KUKA KRL program: ho_st_60301.src, ho_st_60301.dat

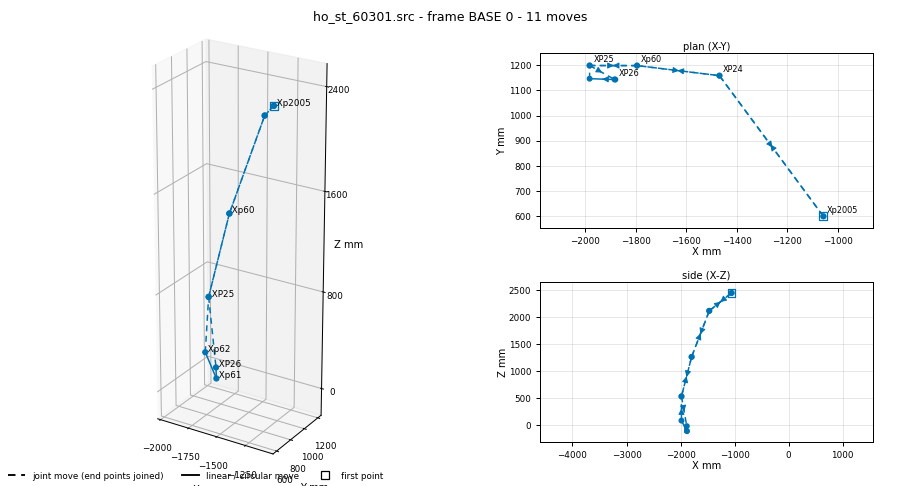
[picture p0: tool path of ho_st_60301.src in frame BASE 0, 11 of 11 moves have a stored position in this frame; points joined in program order, loops and branches not executed]
--- ho_st_60301.src ---
&ACCESS RV2
&REL 251
&COMMENT Busca Peca Frontal Accelo
&PARAM TEMPLATE = C:\KRC\Roboter\Template\vorgabe
&PARAM EDITMASK = *
DEF ho_st_60301( )
;FOLD INI;%{PE}%V3.2.0,%MKUKATPBASIS,%CINIT,%VCOMMON,%P
;FOLD BAS INI;%{E}%V3.2.0,%MKUKATPBASIS,%CINIT,%VINIT,%P
GLOBAL INTERRUPT DECL 3 WHEN $STOPMESS==TRUE DO IR_STOPM ( )
INTERRUPT ON 3
BAS (#INITMOV,0 )
;ENDFOLD (BAS INI)
;FOLD A20 INI;%{E}%V3.2.0,%MKUKATPA20,%CINIT,%VINIT,%P
IF ARC20==TRUE THEN
A20 (ARC_INI)
INTERRUPT DECL 6 WHEN $CYCFLAG[3]==FALSE DO A20(TECH_STOP2)
ENDIF
;ENDFOLD (A20 INI)
;FOLD A10 INI;%{E}%V3.2.0,%MKUKATPARC,%CINIT,%VINIT,%P
IF A10_OPTION==#ACTIVE THEN
INTERRUPT DECL 4 WHEN $CYCFLAG[2]==FALSE DO A10 (#APPL_ERROR)
INTERRUPT DECL 7 WHEN A_ARC_SWI==#ACTIVE DO A10 (#ARC_SEAM)
INTERRUPT DECL 5 WHEN A_FLY_ARC==TRUE DO A10 (#HPU_ARC)
INTERRUPT  ON 5
A10_INI ( )
ENDIF
;ENDFOLD (A10 INI)
;FOLD GRIPPER INI;%{E}%V3.2.0,%MKUKATPGRIPPER,%CINIT,%VINIT,%P
USER_GRP(0,DUMMY,DUMMY,GDEFAULT)
;ENDFOLD (GRIPPER INI)
;FOLD SPOT INI;%{E}%V3.2.0,%MKUKATPSPOT,%CINIT,%VINIT,%P
USERSPOT(#INIT)
;ENDFOLD (SPOT INI)
;FOLD TOUCHSENSE INI;%{E}%V3.2.0,%MKUKATPTS,%CINIT,%VINIT,%P
IF H70_OPTION THEN
INTERRUPT DECL 15 WHEN $MEAS_PULSE[TOUCH_I[TOUCH_ACTIVE].IN_NR] DO H70 (6,CD0 )
INTERRUPT DECL 16 WHEN $ZERO_MOVE DO H70 (7,CD0 )
INTERRUPT DECL 17 WHEN $TECHPAR_C[FG_TOUCH,8]>0.5 DO H70 (8,CD0)
H70 (1,CD0 )
ENDIF
;ENDFOLD (TOUCHSENSE INI)
;FOLD USER INI;%{E}%V3.2.0,%MKUKATPUSER,%CINIT,%VINIT,%P
;Make your modifications here
;ENDFOLD (USER INI)
;ENDFOLD (INI)

; Caracterização dos meios de produção:
; Versão Atual:
; 19/07/2013 12:00 Name: P13.060-R3 CHANGES: Busca Frontal Accelo
; na Geobox

chk_w3_wechs_ok ( )        ;VERIFICAÇÃO DE FERRAMENTA: griper frontal acelo

;FOLD PTP p2005  Vel= 100 % PDAT54 Tool[3]:Gripper Frontal Accelo Base[0];%{PE}%R 4.1.16,%MKUKATPBASIS,%CMOVE,%VPTP,%P 1:PTP, 2:p2005, 3:, 5:100, 7:PDAT54
$BWDSTART = FALSE
PDAT_ACT=PPDAT54
BAS(#PTP_DAT)
FDAT_ACT=Fp2005
BAS(#FRAMES)
BAS(#VEL_PTP,100)
PTP Xp2005
;ENDFOLD

;FOLD OUT 826 'Busca frontal Accelo'  State= TRUE ;%{PE}%R 4.1.16,%MKUKATPBASIS,%COUT,%VOUTX,%P 2:826, 3:'Busca frontal Accelo', 5:TRUE, 6:
$OUT[826]=TRUE
;ENDFOLD
;FOLD OUT 825 'R3 Solic Lib Entrar EST 060 EL_631 '  State= TRUE ;%{PE}%R 4.1.16,%MKUKATPBASIS,%COUT,%VOUTX,%P 2:825, 3:'R3 Solic Lib Entrar EST 060 EL_631 ', 5:TRUE, 6:
$OUT[825]=TRUE
;ENDFOLD
;FOLD WAIT FOR IN 826 'aguarda lib. buscar frontal Accelo'  State= TRUE ;%{PE}%R 4.1.16,%MKUKATPBASIS,%CWAIT_FOR,%VWAIT_FOR,%P 1:0, 2:826, 3:'aguarda lib. buscar frontal Accelo', 5:TRUE, 6:
WAIT FOR $IN[826]==TRUE
;ENDFOLD
;FOLD OUT 826 'Busca frontal Accelo'  State= FALSE ;%{PE}%R 4.1.16,%MKUKATPBASIS,%COUT,%VOUTX,%P 2:826, 3:'Busca frontal Accelo', 5:FALSE, 6:
$OUT[826]=FALSE
;ENDFOLD
;FOLD OUT 825 'R3 Solic Lib Entrar EST 060 EL_631 '  State= FALSE ;%{PE}%R 4.1.16,%MKUKATPBASIS,%COUT,%VOUTX,%P 2:825, 3:'R3 Solic Lib Entrar EST 060 EL_631 ', 5:FALSE, 6:
$OUT[825]=FALSE
;ENDFOLD
;FOLD OUT 846 'R3 solda respot Geo 1 concluida'  State= FALSE ;%{PE}%R 4.1.16,%MKUKATPBASIS,%COUT,%VOUTX,%P 2:846, 3:'R3 solda respot Geo 1 concluida', 5:FALSE, 6:
$OUT[846]=FALSE
;ENDFOLD

;FOLD PTP P24 CONT Vel= 100 % PDAT23 Tool[3]:Gripper Frontal Accelo Base[0];%{PE}%R 4.1.16,%MKUKATPBASIS,%CMOVE,%VPTP,%P 1:PTP, 2:P24, 3:C_PTP, 5:100, 7:PDAT23
$BWDSTART = FALSE
PDAT_ACT=PPDAT23
BAS(#PTP_DAT)
FDAT_ACT=FP24
BAS(#FRAMES)
BAS(#VEL_PTP,100)
PTP XP24 C_PTP
;ENDFOLD
;FOLD PTP p60 CONT Vel= 100 % PDAT41 Tool[3]:Gripper Frontal Accelo Base[0];%{PE}%R 4.1.16,%MKUKATPBASIS,%CMOVE,%VPTP,%P 1:PTP, 2:p60, 3:C_PTP, 5:100, 7:PDAT41
$BWDSTART = FALSE
PDAT_ACT=PPDAT41
BAS(#PTP_DAT)
FDAT_ACT=Fp60
BAS(#FRAMES)
BAS(#VEL_PTP,100)
PTP Xp60 C_PTP
;ENDFOLD
;FOLD PTP P25 CONT Vel= 100 % PDAT24 Tool[3]:Gripper Frontal Accelo Base[0];%{PE}%R 4.1.16,%MKUKATPBASIS,%CMOVE,%VPTP,%P 1:PTP, 2:P25, 3:C_PTP, 5:100, 7:PDAT24
$BWDSTART = FALSE
PDAT_ACT=PPDAT24
BAS(#PTP_DAT)
FDAT_ACT=FP25
BAS(#FRAMES)
BAS(#VEL_PTP,100)
PTP XP25 C_PTP
;ENDFOLD

;FOLD OUT 850 'Area do Operador'  State= FALSE ;%{PE}%R 4.1.16,%MKUKATPBASIS,%COUT,%VOUTX,%P 2:850, 3:'Area do Operador', 5:FALSE, 6:
$OUT[850]=FALSE
;ENDFOLD

;FOLD PTP P26 CONT Vel= 100 % PDAT25 Tool[3]:Gripper Frontal Accelo Base[0];%{PE}%R 4.1.16,%MKUKATPBASIS,%CMOVE,%VPTP,%P 1:PTP, 2:P26, 3:C_PTP, 5:100, 7:PDAT25
$BWDSTART = FALSE
PDAT_ACT=PPDAT25
BAS(#PTP_DAT)
FDAT_ACT=FP26
BAS(#FRAMES)
BAS(#VEL_PTP,100)
PTP XP26 C_PTP
;ENDFOLD

;FOLD ; ponto de pega;%{PE}%R 4.1.16,%MKUKATPBASIS,%CCOMMENT,%VNORMAL,%P 2:ponto de pega
;ENDFOLD
;FOLD LIN p61  Vel= 0.1 m/s CPDAT10 Tool[3]:Gripper Frontal Accelo Base[0];%{PE}%R 4.1.16,%MKUKATPBASIS,%CMOVE,%VLIN,%P 1:LIN, 2:p61, 3:, 5:0.1, 7:CPDAT10
$BWDSTART = FALSE
LDAT_ACT=LCPDAT10
BAS(#CP_DAT)
FDAT_ACT=Fp61
BAS(#FRAMES)
BAS(#VEL_CP,0.1)
LIN Xp61
;ENDFOLD

IF (NOT(GHOST())) THEN
;FOLD WAIT FOR IN 1 'presenca peca1'  State= TRUE ;%{PE}%R 4.1.16,%MKUKATPBASIS,%CWAIT_FOR,%VWAIT_FOR,%P 1:0, 2:1, 3:'presenca peca1', 5:TRUE, 6:
WAIT FOR $IN[1]==TRUE
;ENDFOLD
;FOLD WAIT FOR IN 2 'presenca peca2'  State= TRUE ;%{PE}%R 4.1.16,%MKUKATPBASIS,%CWAIT_FOR,%VWAIT_FOR,%P 1:0, 2:2, 3:'presenca peca2', 5:TRUE, 6:
WAIT FOR $IN[2]==TRUE
;ENDFOLD
ENDIF

;FOLD SET GRP 1  State= CLO  GDAT1;%{PE}%R 4.1.7,%MKUKATPGRP,%CGRP,%VGRP,%P 2:1, 4:2, 5:#NO, 6:GDAT1, 8:0, 10:0
H50(GRP,1,2,GGDAT1)
;ENDFOLD
chk_cilindroZ1_avancado ( )

;FOLD SET GRP 3  State= CLO  GDAT10;%{PE}%R 4.1.7,%MKUKATPGRP,%CGRP,%VGRP,%P 2:3, 4:2, 5:#NO, 6:GDAT10, 8:0, 10:0
H50(GRP,3,2,GGDAT10)
;ENDFOLD
chk_grp03_clo()

;FOLD SET GRP 2  State= CLO  GDAT3;%{PE}%R 4.1.7,%MKUKATPGRP,%CGRP,%VGRP,%P 2:2, 4:2, 5:#NO, 6:GDAT3, 8:0, 10:0
H50(GRP,2,2,GGDAT3)
;ENDFOLD
chk_grp02_clo ( )

;FOLD OUT 828 'Solicita lib. sair magazine'  State= TRUE ;%{PE}%R 4.1.16,%MKUKATPBASIS,%COUT,%VOUTX,%P 2:828, 3:'Solicita lib. sair magazine', 5:TRUE, 6:
$OUT[828]=TRUE
;ENDFOLD
;FOLD WAIT FOR IN 829 'aguarda lib. sair magazine'  State= TRUE ;%{PE}%R 4.1.16,%MKUKATPBASIS,%CWAIT_FOR,%VWAIT_FOR,%P 1:0, 2:829, 3:'aguarda lib. sair magazine', 5:TRUE, 6:
WAIT FOR $IN[829]==TRUE
;ENDFOLD
;FOLD OUT 828 'Solicita lib. sair magazine'  State= FALSE ;%{PE}%R 4.1.16,%MKUKATPBASIS,%COUT,%VOUTX,%P 2:828, 3:'Solicita lib. sair magazine', 5:FALSE, 6:
$OUT[828]=FALSE
;ENDFOLD

;saida com peca
;FOLD LIN p62  Vel= 0.5 m/s CPDAT11 Tool[3]:Gripper Frontal Accelo Base[0];%{PE}%R 4.1.16,%MKUKATPBASIS,%CMOVE,%VLIN,%P 1:LIN, 2:p62, 3:, 5:0.5, 7:CPDAT11
$BWDSTART = FALSE
LDAT_ACT=LCPDAT11
BAS(#CP_DAT)
FDAT_ACT=Fp62
BAS(#FRAMES)
BAS(#VEL_CP,0.5)
LIN Xp62
;ENDFOLD

;FOLD OUT 850 'Area do Operador'  State= TRUE ;%{PE}%R 4.1.16,%MKUKATPBASIS,%COUT,%VOUTX,%P 2:850, 3:'Area do Operador', 5:TRUE, 6:
$OUT[850]=TRUE
;ENDFOLD

;FOLD PTP P27 CONT Vel= 100 % PDAT26 Tool[3]:Gripper Frontal Accelo Base[0];%{PE}%R 4.1.16,%MKUKATPBASIS,%CMOVE,%VPTP,%P 1:PTP, 2:P27, 3:C_PTP, 5:100, 7:PDAT26
$BWDSTART = FALSE
PDAT_ACT=PPDAT26
BAS(#PTP_DAT)
FDAT_ACT=FP27
BAS(#FRAMES)
BAS(#VEL_PTP,100)
PTP XP27 C_PTP
;ENDFOLD
;FOLD PTP P28 CONT Vel= 100 % PDAT27 Tool[3]:Gripper Frontal Accelo Base[0];%{PE}%R 4.1.16,%MKUKATPBASIS,%CMOVE,%VPTP,%P 1:PTP, 2:P28, 3:C_PTP, 5:100, 7:PDAT27
$BWDSTART = FALSE
PDAT_ACT=PPDAT27
BAS(#PTP_DAT)
FDAT_ACT=FP28
BAS(#FRAMES)
BAS(#VEL_PTP,100)
PTP XP28 C_PTP
;ENDFOLD
;FOLD PTP P29 CONT Vel= 100 % PDAT28 Tool[3]:Gripper Frontal Accelo Base[0];%{PE}%R 4.1.16,%MKUKATPBASIS,%CMOVE,%VPTP,%P 1:PTP, 2:P29, 3:C_PTP, 5:100, 7:PDAT28
$BWDSTART = FALSE
PDAT_ACT=PPDAT28
BAS(#PTP_DAT)
FDAT_ACT=FP29
BAS(#FRAMES)
BAS(#VEL_PTP,100)
PTP XP29 C_PTP
;ENDFOLD
;FOLD PTP p2004  Vel= 100 % PDAT53 Tool[3]:Gripper Frontal Accelo Base[0];%{PE}%R 4.1.16,%MKUKATPBASIS,%CMOVE,%VPTP,%P 1:PTP, 2:p2004, 3:, 5:100, 7:PDAT53
$BWDSTART = FALSE
PDAT_ACT=PPDAT53
BAS(#PTP_DAT)
FDAT_ACT=Fp2004
BAS(#FRAMES)
BAS(#VEL_PTP,100)
PTP Xp2004
;ENDFOLD

;FOLD OUT 826 'Busca frontal Accelo'  State= TRUE ;%{PE}%R 4.1.16,%MKUKATPBASIS,%COUT,%VOUTX,%P 2:826, 3:'Busca frontal Accelo', 5:TRUE, 6:
$OUT[826]=TRUE
;ENDFOLD
;FOLD PULSE 829 'Pegou peca'  State= TRUE   Time= 3 sec;%{PE}%R 4.1.16,%MKUKATPBASIS,%COUT,%VPULSE,%P 2:829, 3:'Pegou peca', 5:TRUE, 6:, 8:3
PULSE($OUT[829], TRUE,3)
;ENDFOLD

;FOLD WAIT FOR IN 179 'protecao da pinca aberto'  State= FALSE ;%{PE}%R 4.1.16,%MKUKATPBASIS,%CWAIT_FOR,%VWAIT_FOR,%P 1:0, 2:179, 3:'protecao da pinca aberto', 5:FALSE, 6:
WAIT FOR $IN[179]==FALSE
;ENDFOLD
;FOLD WAIT FOR IN 180 'protecao da pinca fechado'  State= TRUE ;%{PE}%R 4.1.16,%MKUKATPBASIS,%CWAIT_FOR,%VWAIT_FOR,%P 1:0, 2:180, 3:'protecao da pinca fechado', 5:TRUE, 6:
WAIT FOR $IN[180]==TRUE
;ENDFOLD

END

--- ho_st_60301.dat ---
&ACCESS RV2
&REL 251
&COMMENT Busca Peca Frontal Accelo
&PARAM TEMPLATE = C:\KRC\Roboter\Template\vorgabe
&PARAM EDITMASK = *
DEFDAT  HO_ST_60301
;FOLD EXTERNAL DECLARATIONS;%{PE}%V3.2.0,%MKUKATPBASIS,%CEXT,%VCOMMON,%P
;FOLD BAS EXT;%{PE}%V3.2.0,%MKUKATPBASIS,%CEXT,%VEXT,%P
EXT  BAS (BAS_COMMAND  :IN,REAL  :IN )
DECL INT SUCCESS
;ENDFOLD
;FOLD A10 EXT;%{E}%V3.2.0,%MKUKATPARC,%CEXT,%VEXT,%P
EXT  A10 (A_CMD_T  :IN,A_STRT_T  :IN,A_WELD_T  :IN,A_END_T  :IN,INT  :IN )
;ENDFOLD
;FOLD A20 EXT;%{E}%V3.2.0,%MKUKATPA20,%CEXT,%VEXT,%P
EXT  A20 (INT  :IN,WELD_ST  :IN,WELD_FI  :IN,INT  :IN )
;ENDFOLD
;FOLD GRIPPER EXT;%{E}%V3.2.0,%MKUKATPGRIPPER,%CEXT,%VEXT,%P
EXT  H50 (INT  :IN,INT  :IN,INT  :IN,GRP_TYP  :IN )
;ENDFOLD
;FOLD SPOT EXT;%{E}%V3.2.0,%MKUKATPSPOT,%CEXT,%VEXT,%P
EXT  USERSPOT (S_COMMAND  :IN,SPOT_TYPE  :IN )
;ENDFOLD
;FOLD TOUCHSENSE EXT;%{E}%V3.2.0,%MKUKATPTS,%CEXT,%VEXT,%P
EXT  H70 (INT  :IN,SRCH_TYP_2  :OUT,E6POS  :IN,SRCH_TYP_3  :IN,SRCH_TYP_2  :IN,SRCH_TYP_2  :IN,SRCH_TYP_2  :IN,SRCH_TYP_2  :IN,SRCH_TYP_2  :IN,INT  :IN )
;ENDFOLD
;FOLD USER EXT;%{E}%V3.2.0,%MKUKATPUSER,%CEXT,%VEXT,%P
;Make here your modifications
;ENDFOLD
;ENDFOLD

DECL BASIS_SUGG_T LAST_BASIS={POINT1[] "p2005                   ",POINT2[] "p2005                   ",CP_PARAMS[] "CPDAT18                 ",PTP_PARAMS[] "PDAT54                  ",CONT[] "                        ",CP_VEL[] "0.2                     ",PTP_VEL[] "50                      "}
DECL E6POS XP1={x -188.3992,y 2368.7981,z 816.157471,a 0.682591379,b 56.9728508,c -155.483307,s 6,t 51,e1 0.0,e2 0.0,e3 0.0,e4 0.0,e5 0.0,e6 0.0}


DECL FDAT FP1={TOOL_NO 8,BASE_NO 0,IPO_FRAME #BASE}
DECL PDAT PPDAT1={VEL 100.0,ACC 100.0,APO_DIST 100.0}
DECL E6POS XP2={x 39.6335411,y 2248.2561,z 963.446594,a 0.683832824,b 56.9725304,c -155.481995,s 6,t 51,e1 0.0,e2 0.0,e3 0.0,e4 0.0,e5 0.0,e6 0.0}
DECL FDAT FP2={TOOL_NO 8,BASE_NO 0,IPO_FRAME #BASE}
DECL PDAT PPDAT2={VEL 100.0,ACC 100.0,APO_DIST 100.0}
DECL E6POS XP3={x 388.941711,y 1754.29297,z 2068.00708,a 129.908005,b 79.1631622,c 52.0251884,s 2,t 35,e1 0.0,e2 0.0,e3 0.0,e4 0.0,e5 0.0,e6 0.0}
DECL FDAT FP3={TOOL_NO 8,BASE_NO 0,IPO_FRAME #BASE}
DECL PDAT PPDAT3={VEL 100.0,ACC 100.0,APO_DIST 100.0}
DECL E6POS XP4={x -141.421799,y 2321.63794,z 903.706726,a -12.8919296,b 56.8668289,c -155.093994,s 6,t 51,e1 0.0,e2 0.0,e3 0.0,e4 0.0,e5 0.0,e6 0.0}

DECL FDAT FP4={TOOL_NO 8,BASE_NO 0,IPO_FRAME #BASE}
DECL PDAT PPDAT4={VEL 100.0,ACC 100.0,APO_DIST 100.0}
DECL E6POS XP5={x -310.951813,y 2507.78101,z 762.400391,a -5.76357794,b 56.6388206,c -155.210098,s 6,t 51,e1 0.0,e2 0.0,e3 0.0,e4 0.0,e5 0.0,e6 0.0}
DECL FDAT FP5={TOOL_NO 8,BASE_NO 0,IPO_FRAME #BASE}
DECL PDAT PPDAT5={VEL 100.0,ACC 100.0,APO_DIST 100.0}
DECL E6POS XP6={x -231.908905,y 2732.73511,z 874.473572,a 62.2883606,b -0.0793622211,c -89.9837265,s 6,t 51,e1 0.0,e2 0.0,e3 0.0,e4 0.0,e5 0.0,e6 0.0}
DECL FDAT FP6={TOOL_NO 3,BASE_NO 0,IPO_FRAME #BASE}
DECL PDAT PPDAT6={VEL 100.0,ACC 100.0,APO_DIST 100.0}
DECL E6POS XP7={x -138.7957,y 2749.80103,z 865.714417,a 64.2388,b -0.0770005435,c -89.9825897,s 6,t 51,e1 0.0,e2 0.0,e3 0.0,e4 0.0,e5 0.0,e6 0.0}
DECL FDAT FP7={TOOL_NO 3,BASE_NO 0,IPO_FRAME #BASE}
DECL PDAT PPDAT7={VEL 100.0,ACC 100.0,APO_DIST 100.0}
DECL E6POS XP8={x -58.7346306,y 2732.94092,z 865.675293,a 67.7668915,b -0.075337939,c -89.9879227,s 6,t 51,e1 0.0,e2 0.0,e3 0.0,e4 0.0,e5 0.0,e6 0.0}
DECL FDAT FP8={TOOL_NO 3,BASE_NO 0,IPO_FRAME #BASE}
DECL PDAT PPDAT8={VEL 100.0,ACC 100.0,APO_DIST 100.0}
DECL E6POS XP9={x -4.80422878,y 2723.65308,z 865.806519,a 69.4628601,b -0.0796707496,c -89.9865265,s 6,t 51,e1 0.0,e2 0.0,e3 0.0,e4 0.0,e5 0.0,e6 0.0}
DECL FDAT FP9={TOOL_NO 3,BASE_NO 0,IPO_FRAME #BASE}
DECL PDAT PPDAT9={VEL 100.0,ACC 100.0,APO_DIST 100.0}
DECL E6POS XP10={x 96.421463,y 2705.94312,z 852.752686,a 59.7485199,b -0.0976489186,c -89.969368,s 6,t 51,e1 0.0,e2 0.0,e3 0.0,e4 0.0,e5 0.0,e6 0.0}
DECL FDAT FP10={TOOL_NO 3,BASE_NO 0,IPO_FRAME #BASE}
DECL PDAT PPDAT10={VEL 100.0,ACC 100.0,APO_DIST 100.0}
DECL E6POS XP11={x 254.399094,y 2660.85889,z 851.276611,a 47.4197311,b -0.094424963,c -89.9508286,s 6,t 51,e1 0.0,e2 0.0,e3 0.0,e4 0.0,e5 0.0,e6 0.0}
DECL FDAT FP11={TOOL_NO 3,BASE_NO 0,IPO_FRAME #BASE}
DECL PDAT PPDAT11={VEL 100.0,ACC 100.0,APO_DIST 100.0}
DECL E6POS XP12={x 254.197098,y 2660.07202,z 1289.99695,a 47.4186096,b -0.0936179385,c -90.4839935,s 6,t 51,e1 0.0,e2 0.0,e3 0.0,e4 0.0,e5 0.0,e6 0.0}
DECL FDAT FP12={TOOL_NO 3,BASE_NO 0,IPO_FRAME #BASE}
DECL PDAT PPDAT12={VEL 100.0,ACC 100.0,APO_DIST 100.0}
DECL E6POS XP13={x 387.00351,y 2537.04199,z 1725.88306,a 47.4178085,b -0.0868179128,c -81.4952316,s 6,t 51,e1 0.0,e2 0.0,e3 0.0,e4 0.0,e5 0.0,e6 0.0}
DECL FDAT FP13={TOOL_NO 3,BASE_NO 0,IPO_FRAME #BASE}
DECL PDAT PPDAT13={VEL 100.0,ACC 100.0,APO_DIST 100.0}
DECL E6POS XP14={x 577.404114,y 2286.39795,z 1935.52197,a 30.7294006,b 4.42975616,c -75.2716522,s 6,t 51,e1 0.0,e2 0.0,e3 0.0,e4 0.0,e5 0.0,e6 0.0}
DECL FDAT FP14={TOOL_NO 3,BASE_NO 0,IPO_FRAME #BASE}
DECL PDAT PPDAT14={VEL 100.0,ACC 100.0,APO_DIST 100.0}
DECL E6POS XP15={x -210.601395,y 2793.87988,z 858.125427,a 47.6891098,b -0.311072499,c -90.0127563,s 6,t 51,e1 0.0,e2 0.0,e3 0.0,e4 0.0,e5 0.0,e6 0.0}
DECL FDAT FP15={TOOL_NO 3,BASE_NO 0,IPO_FRAME #BASE}
DECL PDAT PPDAT15={VEL 100.0,ACC 100.0,APO_DIST 100.0}
DECL LDAT LCPDAT1={VEL 2.0,ACC 100.0,APO_DIST 100.0,APO_FAC 50.0}
DECL E6POS XP16={x -253.589203,y 2420.03198,z 826.688293,a -15.0486002,b 56.5221214,c -156.482697,s 6,t 51,e1 0.0,e2 0.0,e3 0.0,e4 0.0,e5 0.0,e6 0.0}
DECL FDAT FP16={TOOL_NO 8,BASE_NO 0,IPO_FRAME #BASE}
DECL LDAT LCPDAT2={VEL 2.0,ACC 100.0,APO_DIST 100.0,APO_FAC 50.0}
DECL LDAT LCPDAT3={VEL 2.0,ACC 100.0,APO_DIST 100.0,APO_FAC 50.0}
DECL E6POS XP17={x -104.003502,y 2593.61499,z 862.898682,a 47.8507004,b -0.443317294,c -89.9662323,s 6,t 51,e1 0.0,e2 0.0,e3 0.0,e4 0.0,e5 0.0,e6 0.0}
DECL FDAT FP17={TOOL_NO 3,BASE_NO 0,IPO_FRAME #BASE}
DECL PDAT PPDAT16={VEL 100.0,ACC 100.0,APO_DIST 100.0}
DECL E6POS XP18={x -114.378899,y 2558.99609,z 1228.50195,a 42.74683,b -0.281747609,c -89.6939468,s 6,t 51,e1 0.0,e2 0.0,e3 0.0,e4 0.0,e5 0.0,e6 0.0}
DECL FDAT FP18={TOOL_NO 3,BASE_NO 0,IPO_FRAME #BASE}
DECL PDAT PPDAT17={VEL 100.0,ACC 100.0,APO_DIST 100.0}
DECL E6POS XP19={x 59.8382301,y 2366.573,z 1678.95105,a 32.0545197,b 2.27294707,c -77.4810028,s 6,t 51,e1 0.0,e2 0.0,e3 0.0,e4 0.0,e5 0.0,e6 0.0}
DECL FDAT FP19={TOOL_NO 3,BASE_NO 0,IPO_FRAME #BASE}
DECL PDAT PPDAT18={VEL 100.0,ACC 100.0,APO_DIST 100.0}
DECL E6POS XP20={x 178.339905,y 2018.22302,z 1695.13098,a 16.4725895,b 3.63115811,c -69.0822067,s 6,t 51,e1 0.0,e2 0.0,e3 0.0,e4 0.0,e5 0.0,e6 0.0}
DECL FDAT FP20={TOOL_NO 3,BASE_NO 0,IPO_FRAME #BASE}
DECL PDAT PPDAT19={VEL 100.0,ACC 100.0,APO_DIST 100.0}
DECL E6POS XP21={x 103.363403,y 1772.48596,z 1818.14697,a 12.0467701,b 4.32170582,c -60.2828217,s 6,t 51,e1 0.0,e2 0.0,e3 0.0,e4 0.0,e5 0.0,e6 0.0}
DECL FDAT FP21={TOOL_NO 3,BASE_NO 0,IPO_FRAME #BASE}
DECL PDAT PPDAT20={VEL 100.0,ACC 100.0,APO_DIST 100.0}
DECL E6POS XP22={x 2104.2251,y 68.1197662,z 102.1996,a -0.666801214,b -0.144442394,c -152.486694,s 2,t 3,e1 0.0,e2 0.0,e3 0.0,e4 0.0,e5 0.0,e6 0.0}
DECL FDAT FP22={TOOL_NO 3,BASE_NO 0,IPO_FRAME #BASE}
DECL PDAT PPDAT21={VEL 100.0,ACC 100.0,APO_DIST 100.0}
DECL E6POS XP23={x -1056.99194,y 600.572815,z 2451.80591,a 175.843597,b -72.5620575,c 179.205307,s 2,t 3,e1 0.0,e2 0.0,e3 0.0,e4 0.0,e5 0.0,e6 0.0}
DECL FDAT FP23={TOOL_NO 3,BASE_NO 0,IPO_FRAME #BASE}
DECL PDAT PPDAT22={VEL 100.0,ACC 80.0,APO_DIST 3.0}
DECL E6POS XP24={x -1468.95703,y 1158.19897,z 2120.92505,a 177.713699,b -54.6900291,c 178.097107,s 2,t 11,e1 0.0,e2 0.0,e3 0.0,e4 0.0,e5 0.0,e6 0.0}
DECL FDAT FP24={TOOL_NO 3,BASE_NO 0,IPO_FRAME #BASE}
DECL PDAT PPDAT23={VEL 100.0,ACC 100.0,APO_DIST 50.0}
DECL E6POS XP25={x -1983.53406,y 1198.328,z 537.303406,a 179.117096,b 7.47287893,c -179.832199,s 2,t 3,e1 0.0,e2 0.0,e3 0.0,e4 0.0,e5 0.0,e6 0.0}
DECL FDAT FP25={TOOL_NO 3,BASE_NO 0,IPO_FRAME #BASE}
DECL PDAT PPDAT24={VEL 100.0,ACC 100.0,APO_DIST 50.0}
DECL E6POS XP26={x -1884.86902,y 1143.23401,z -12.8902597,a 178.553894,b 27.9167995,c -179.580795,s 2,t 3,e1 0.0,e2 0.0,e3 0.0,e4 0.0,e5 0.0,e6 0.0}
DECL FDAT FP26={TOOL_NO 3,BASE_NO 0,IPO_FRAME #BASE}
DECL PDAT PPDAT25={VEL 100.0,ACC 100.0,APO_DIST 20.0}
DECL E6POS XP27={x -1983.52502,y 1198.323,z 537.230286,a 179.116501,b 7.47453594,c -179.831207,s 2,t 3,e1 0.0,e2 0.0,e3 0.0,e4 0.0,e5 0.0,e6 0.0}
DECL FDAT FP27={TOOL_NO 3,BASE_NO 0,IPO_FRAME #BASE}
DECL PDAT PPDAT26={VEL 100.0,ACC 100.0,APO_DIST 20.0}
DECL E6POS XP28={x -1795.58105,y 1198.05896,z 1268.58801,a 179.125305,b -28.5398693,c -179.794601,s 2,t 3,e1 0.0,e2 0.0,e3 0.0,e4 0.0,e5 0.0,e6 0.0}
DECL FDAT FP28={TOOL_NO 3,BASE_NO 0,IPO_FRAME #BASE}
DECL PDAT PPDAT27={VEL 100.0,ACC 100.0,APO_DIST 20.0}
DECL E6POS XP29={x -1468.95703,y 1158.19397,z 2120.92896,a 177.714005,b -54.690239,c 178.096802,s 2,t 11,e1 0.0,e2 0.0,e3 0.0,e4 0.0,e5 0.0,e6 0.0}
DECL FDAT FP29={TOOL_NO 3,BASE_NO 0,IPO_FRAME #BASE}
DECL PDAT PPDAT28={VEL 100.0,ACC 100.0,APO_DIST 20.0}
DECL E6POS XP30={x 103.363403,y 1772.48596,z 1818.14697,a 12.0467701,b 4.32170582,c -60.2828217,s 6,t 51,e1 0.0,e2 0.0,e3 0.0,e4 0.0,e5 0.0,e6 0.0}
DECL FDAT FP30={TOOL_NO 3,BASE_NO 0,IPO_FRAME #BASE}
DECL PDAT PPDAT29={VEL 100.0,ACC 100.0,APO_DIST 100.0}
DECL E6POS XP31={x 178.339905,y 2018.22302,z 1695.13098,a 16.4725895,b 3.63115811,c -69.0822067,s 6,t 51,e1 0.0,e2 0.0,e3 0.0,e4 0.0,e5 0.0,e6 0.0}
DECL FDAT FP31={TOOL_NO 3,BASE_NO 0,IPO_FRAME #BASE}
DECL PDAT PPDAT30={VEL 100.0,ACC 100.0,APO_DIST 100.0}
DECL E6POS XP32={x 59.8382301,y 2366.573,z 1678.95105,a 32.0545197,b 2.27294707,c -77.4810028,s 6,t 51,e1 0.0,e2 0.0,e3 0.0,e4 0.0,e5 0.0,e6 0.0}
DECL FDAT FP32={TOOL_NO 3,BASE_NO 0,IPO_FRAME #BASE}
DECL PDAT PPDAT31={VEL 100.0,ACC 100.0,APO_DIST 100.0}
DECL E6POS XP33={x -114.378899,y 2558.99609,z 1228.50195,a 42.74683,b -0.281747609,c -89.6939468,s 6,t 51,e1 0.0,e2 0.0,e3 0.0,e4 0.0,e5 0.0,e6 0.0}
DECL FDAT FP33={TOOL_NO 3,BASE_NO 0,IPO_FRAME #BASE}
DECL PDAT PPDAT32={VEL 100.0,ACC 100.0,APO_DIST 100.0}
DECL E6POS XP34={x -69.7102814,y 2637.021,z 863.732788,a 46.0948906,b -0.300397307,c -89.7107086,s 6,t 51,e1 0.0,e2 0.0,e3 0.0,e4 0.0,e5 0.0,e6 0.0}
DECL FDAT FP34={TOOL_NO 3,BASE_NO 0,IPO_FRAME #BASE}
DECL PDAT PPDAT33={VEL 100.0,ACC 100.0,APO_DIST 100.0}
DECL E6POS XP35={x -217.495407,y 2798.87402,z 862.13623,a 47.7863503,b -0.181169301,c -89.6277924,s 6,t 51,e1 0.0,e2 0.0,e3 0.0,e4 0.0,e5 0.0,e6 0.0}
DECL FDAT FP35={TOOL_NO 3,BASE_NO 0,IPO_FRAME #BASE}
DECL PDAT PPDAT34={VEL 100.0,ACC 100.0,APO_DIST 100.0}
DECL E6POS XP36={x -217.537292,y 2799.2251,z 752.995728,a 48.2843094,b -0.3213332,c -89.7200928,s 6,t 51,e1 0.0,e2 0.0,e3 0.0,e4 0.0,e5 0.0,e6 0.0}
DECL FDAT FP36={TOOL_NO 3,BASE_NO 0,IPO_FRAME #BASE}
DECL LDAT LCPDAT4={VEL 2.0,ACC 100.0,APO_DIST 100.0,APO_FAC 50.0}
DECL E6POS XP37={x -218.973099,y 2799.72998,z 833.772522,a 48.4467506,b -0.344602793,c -89.9268036,s 6,t 51,e1 0.0,e2 0.0,e3 0.0,e4 0.0,e5 0.0,e6 0.0}
DECL FDAT FP37={TOOL_NO 3,BASE_NO 0,IPO_FRAME #BASE}
DECL LDAT LCPDAT5={VEL 2.0,ACC 100.0,APO_DIST 100.0,APO_FAC 50.0}
DECL E6POS XP38={x -334.715088,y 2494.78711,z 762.013611,a -15.0434103,b 56.5220718,c -156.471695,s 6,t 51,e1 0.0,e2 0.0,e3 0.0,e4 0.0,e5 0.0,e6 0.0}
DECL FDAT FP38={TOOL_NO 8,BASE_NO 0,IPO_FRAME #BASE}
DECL LDAT LCPDAT6={VEL 2.0,ACC 100.0,APO_DIST 100.0,APO_FAC 50.0}
DECL E6POS XP39={x 2135.1189,y 879.29187,z 1623.97302,a 95.7743378,b -6.67306614,c 140.607193,s 2,t 3,e1 0.0,e2 0.0,e3 0.0,e4 0.0,e5 0.0,e6 0.0}
DECL FDAT FP39={TOOL_NO 3,BASE_NO 0,IPO_FRAME #BASE}
DECL PDAT PPDAT35={VEL 100.0,ACC 100.0,APO_DIST 100.0}
DECL E6POS XP40={x 2290.56299,y -695.490601,z 1091.52795,a 74.2140274,b 81.0776062,c 153.915894,s 2,t 2,e1 0.0,e2 0.0,e3 0.0,e4 0.0,e5 0.0,e6 0.0}
DECL FDAT FP40={TOOL_NO 3,BASE_NO 0,IPO_FRAME #BASE}
DECL PDAT PPDAT36={VEL 100.0,ACC 100.0,APO_DIST 100.0}
DECL E6POS XP41={x 2120.95801,y -1006.67102,z 519.729919,a 146.695801,b 89.4882584,c -122.776802,s 2,t 2,e1 0.0,e2 0.0,e3 0.0,e4 0.0,e5 0.0,e6 0.0}
DECL FDAT FP41={TOOL_NO 3,BASE_NO 0,IPO_FRAME #BASE}
DECL PDAT PPDAT37={VEL 100.0,ACC 100.0,APO_DIST 100.0}
DECL E6POS XP42={x 2103.9519,y -1494.86694,z 502.313507,a -90.9648972,b 89.7392731,c -0.781405687,s 2,t 2,e1 0.0,e2 0.0,e3 0.0,e4 0.0,e5 0.0,e6 0.0}
DECL FDAT FP42={TOOL_NO 3,BASE_NO 0,IPO_FRAME #BASE}
DECL PDAT PPDAT38={VEL 100.0,ACC 100.0,APO_DIST 100.0}
DECL E6POS XP43={x 2103.896,y -1542.37903,z 502.545013,a -91.1217804,b 89.7371826,c -0.941302776,s 2,t 2,e1 0.0,e2 0.0,e3 0.0,e4 0.0,e5 0.0,e6 0.0}
DECL FDAT FP43={TOOL_NO 3,BASE_NO 0,IPO_FRAME #BASE}
DECL LDAT LCPDAT7={VEL 2.0,ACC 100.0,APO_DIST 100.0,APO_FAC 50.0}
DECL E6POS XP44={x 2105.36499,y -1049.36401,z 552.007874,a -90.6014099,b 89.7380829,c -0.414461106,s 2,t 2,e1 0.0,e2 0.0,e3 0.0,e4 0.0,e5 0.0,e6 0.0}
DECL FDAT FP44={TOOL_NO 3,BASE_NO 0,IPO_FRAME #BASE}
DECL PDAT PPDAT39={VEL 100.0,ACC 100.0,APO_DIST 100.0}
DECL E6POS XTESTE={x -218.994202,y 2799.72998,z 855.550476,a 48.4468689,b -0.344231814,c -89.9264526,s 6,t 51,e1 0.0,e2 0.0,e3 0.0,e4 0.0,e5 0.0,e6 0.0}
DECL FDAT Fteste={TOOL_NO 3,BASE_NO 0,IPO_FRAME #BASE}
DECL LDAT LCPDAT8={VEL 2.0,ACC 100.0,APO_DIST 100.0,APO_FAC 50.0}
DECL E6POS XP200={x -318.375702,y 2479.64697,z 775.077576,a -15.0468197,b 56.522541,c -156.479507,s 6,t 51,e1 0.0,e2 0.0,e3 0.0,e4 0.0,e5 0.0,e6 0.0}
DECL FDAT Fp200={TOOL_NO 8,BASE_NO 0,IPO_FRAME #BASE}
DECL LDAT LCPDAT9={VEL 2.0,ACC 100.0,APO_DIST 100.0,APO_FAC 50.0}
DECL PDAT PPDAT40={VEL 100.0,ACC 100.0,APO_DIST 100.0}
DECL E6POS XP60={x -1795.57996,y 1198.06104,z 1268.58301,a 179.124603,b -28.5397491,c -179.794098,s 2,t 3,e1 0.0,e2 0.0,e3 0.0,e4 0.0,e5 0.0,e6 0.0}
DECL FDAT Fp60={TOOL_NO 3,BASE_NO 0,IPO_FRAME #BASE}
DECL PDAT PPDAT41={VEL 100.0,ACC 100.0,APO_DIST 50.0}
DECL E6POS XP61={x -1881.53406,y 1142.78101,z -106.679398,a 178.040802,b 28.7168198,c -179.987198,s 2,t 3,e1 0.0,e2 0.0,e3 0.0,e4 0.0,e5 0.0,e6 0.0}
DECL FDAT Fp61={TOOL_NO 3,BASE_NO 0,IPO_FRAME #BASE}
DECL LDAT LCPDAT10={VEL 2.0,ACC 100.0,APO_DIST 100.0,APO_FAC 50.0}
DECL GRP_SUGG_T LAST_GRP={NUMBER[] "3                       ",STATE[] "1                       ",PARAMS[] "GDAT14                  "}
DECL GRP_TYP GCONT={G_APO #YES,TIME 0.0,CTRL #OFF,DLY 0,DST 0}
DECL GRP_TYP GGDAT0={G_APO #NO,TIME 0.200000003,CTRL #OFF,DLY 0,DST 1}
DECL GRP_TYP GGDAT1={G_APO #NO,TIME 0.200000003,CTRL #OFF,DLY 0,DST 1}
DECL GRP_TYP GGDAT2={G_APO #NO,TIME 0.200000003,CTRL #OFF,DLY 0,DST 1}
DECL GRP_TYP GGDAT3={G_APO #NO,TIME 0.200000003,CTRL #OFF,DLY 0,DST 1}
DECL GRP_TYP GGDAT4={G_APO #NO,TIME 0.200000003,CTRL #OFF,DLY 0,DST 1}
DECL FDAT FHOME1={TOOL_NO 3,BASE_NO 0,IPO_FRAME #BASE}
DECL E6POS XP62={x -1983.52905,y 1146.19604,z 89.4334183,a 178.555099,b 28.1790791,c -179.753906,s 2,t 3,e1 0.0,e2 0.0,e3 0.0,e4 0.0,e5 0.0,e6 0.0}
DECL FDAT Fp62={TOOL_NO 3,BASE_NO 0,IPO_FRAME #BASE}
DECL LDAT LCPDAT11={VEL 2.0,ACC 100.0,APO_DIST 5.0,APO_FAC 50.0}
DECL PDAT PPDAT42={VEL 100.0,ACC 100.0,APO_DIST 3.0}
DECL PDAT PPDAT43={VEL 100.0,ACC 100.0,APO_DIST 100.0}
DECL FDAT FHOME2={TOOL_NO 3,BASE_NO 0,IPO_FRAME #BASE}
DECL PDAT PPDAT44={VEL 100.0,ACC 100.0,APO_DIST 100.0}
DECL GRP_TYP GGDAT5={G_APO #NO,TIME 0.200000003,CTRL #OFF,DLY 0,DST 1}
DECL GRP_TYP GGDAT6={G_APO #NO,TIME 0.200000003,CTRL #OFF,DLY 0,DST 1}
DECL E6POS XP300={x 2103.87793,y -1542.31702,z 502.337585,a -91.9767227,b 89.7423706,c -1.79670501,s 2,t 2,e1 0.0,e2 0.0,e3 0.0,e4 0.0,e5 0.0,e6 0.0}
DECL FDAT Fp300={TOOL_NO 3,BASE_NO 0,IPO_FRAME #BASE}
DECL PDAT PPDAT45={VEL 100.0,ACC 100.0,APO_DIST 100.0}
DECL E6POS XP301={x 2101.01196,y -1428.62,z 807.025513,a 29.7582302,b 15.1351204,c 89.7658234,s 2,t 2,e1 0.0,e2 0.0,e3 0.0,e4 0.0,e5 0.0,e6 0.0}
DECL FDAT Fp301={TOOL_NO 8,BASE_NO 0,IPO_FRAME #BASE}
DECL PDAT PPDAT46={VEL 100.0,ACC 100.0,APO_DIST 100.0}
DECL E6POS XP302={x 1998.20703,y -1249.63599,z 806.080017,a 29.7583504,b 15.1435204,c 89.7742615,s 2,t 2,e1 0.0,e2 0.0,e3 0.0,e4 0.0,e5 0.0,e6 0.0}
DECL FDAT Fp302={TOOL_NO 8,BASE_NO 0,IPO_FRAME #BASE}
DECL LDAT LCPDAT12={VEL 2.0,ACC 100.0,APO_DIST 100.0,APO_FAC 50.0}
DECL E6POS XP303={x 1998.20703,y -1249.63599,z 806.080017,a 29.7583504,b 15.1435204,c 89.7742615,s 2,t 2,e1 0.0,e2 0.0,e3 0.0,e4 0.0,e5 0.0,e6 0.0}
DECL FDAT Fp303={TOOL_NO 8,BASE_NO 0,IPO_FRAME #BASE}
DECL LDAT LCPDAT13={VEL 2.0,ACC 100.0,APO_DIST 100.0,APO_FAC 50.0}
DECL E6POS XP304={x 1705.78699,y -739.28833,z 803.88092,a 29.7551403,b 15.1431599,c 89.7668915,s 2,t 2,e1 0.0,e2 0.0,e3 0.0,e4 0.0,e5 0.0,e6 0.0}
DECL FDAT Fp304={TOOL_NO 8,BASE_NO 0,IPO_FRAME #BASE}
DECL PDAT PPDAT47={VEL 100.0,ACC 100.0,APO_DIST 100.0}
DECL E6POS XP305={x -215.8284,y 2796.93311,z 843.476013,a 47.9605103,b 0.0409639515,c -90.3939896,s 6,t 51,e1 0.0,e2 0.0,e3 0.0,e4 0.0,e5 0.0,e6 0.0}
DECL FDAT Fp305={TOOL_NO 3,BASE_NO 0,IPO_FRAME #BASE}
DECL LDAT LCPDAT15={VEL 2.0,ACC 100.0,APO_DIST 100.0,APO_FAC 50.0}
DECL E6POS XP306={x -92.6007004,y 2685.50098,z 861.002319,a 47.788929,b -0.179067105,c -89.6297226,s 6,t 51,e1 0.0,e2 0.0,e3 0.0,e4 0.0,e5 0.0,e6 0.0}
DECL FDAT Fp306={TOOL_NO 3,BASE_NO 0,IPO_FRAME #BASE}
DECL LDAT LCPDAT16={VEL 2.0,ACC 100.0,APO_DIST 100.0,APO_FAC 50.0}
DECL E6POS XP307={x -215.8311,y 2796.93311,z 760.875671,a 47.960289,b 0.0413109697,c -90.3944168,s 6,t 51,e1 0.0,e2 0.0,e3 0.0,e4 0.0,e5 0.0,e6 0.0}
DECL FDAT Fp307={TOOL_NO 3,BASE_NO 0,IPO_FRAME #BASE}
DECL LDAT LCPDAT17={VEL 2.0,ACC 100.0,APO_DIST 100.0,APO_FAC 50.0}
DECL E6POS XP308={x -249.264603,y 2416.05396,z 831.613281,a -13.6855202,b 56.5440903,c -155.689804,s 6,t 51,e1 0.0,e2 0.0,e3 0.0,e4 0.0,e5 0.0,e6 0.0}
DECL FDAT Fp308={TOOL_NO 8,BASE_NO 0,IPO_FRAME #BASE}
DECL LDAT LCPDAT18={VEL 2.0,ACC 100.0,APO_DIST 100.0,APO_FAC 50.0}
DECL PDAT PPDAT48={VEL 100.0,ACC 100.0,APO_DIST 100.0}
DECL E6POS XP2000={x 14.7387199,y 2430.83203,z 1561.30005,a 44.1596794,b -0.293628901,c -80.8446121,s 6,t 51,e1 0.0,e2 0.0,e3 0.0,e4 0.0,e5 0.0,e6 0.0}
DECL FDAT Fp2000={TOOL_NO 3,BASE_NO 0,IPO_FRAME #BASE}
DECL PDAT PPDAT49={VEL 100.0,ACC 100.0,APO_DIST 100.0}
DECL E6POS XP2001={x -207.498093,y 2790.38208,z 871.288025,a 47.096241,b 0.0432586595,c -89.4638367,s 6,t 51,e1 0.0,e2 0.0,e3 0.0,e4 0.0,e5 0.0,e6 0.0}
DECL FDAT Fp2001={TOOL_NO 3,BASE_NO 0,IPO_FRAME #BASE}
DECL PDAT PPDAT50={VEL 100.0,ACC 100.0,APO_DIST 100.0}
DECL E6POS XP2002={x -28.5181293,y 2384.37012,z 1449.54504,a 37.3302917,b 0.506031811,c -84.0773773,s 6,t 51,e1 0.0,e2 0.0,e3 0.0,e4 0.0,e5 0.0,e6 0.0}
DECL FDAT Fp2002={TOOL_NO 3,BASE_NO 0,IPO_FRAME #BASE}
DECL PDAT PPDAT51={VEL 100.0,ACC 100.0,APO_DIST 100.0}
DECL GRP_TYP GGDAT7={G_APO #NO,TIME 0.200000003,CTRL #OFF,DLY 0,DST 1}
DECL GRP_TYP GGDAT8={G_APO #NO,TIME 0.200000003,CTRL #OFF,DLY 0,DST 1}
DECL GRP_TYP GGDAT9={G_APO #NO,TIME 0.200000003,CTRL #OFF,DLY 0,DST 1}
DECL GRP_TYP GGDAT10={G_APO #NO,TIME 0.200000003,CTRL #OFF,DLY 0,DST 1}
DECL E6POS XP2003={x -1885.86499,y 1144.86401,z -103.444,a 178.647202,b 28.0053997,c -179.457993,s 2,t 3,e1 0.0,e2 0.0,e3 0.0,e4 0.0,e5 0.0,e6 0.0}
DECL FDAT Fp2003={TOOL_NO 3,BASE_NO 0,IPO_FRAME #BASE}
DECL PDAT PPDAT52={VEL 100.0,ACC 100.0,APO_DIST 100.0}
DECL GRP_TYP GGDAT11={G_APO #NO,TIME 0.200000003,CTRL #OFF,DLY 0,DST 1}
DECL GRP_TYP GGDAT12={G_APO #NO,TIME 0.200000003,CTRL #OFF,DLY 0,DST 1}
DECL GRP_TYP GGDAT13={G_APO #NO,TIME 0.200000003,CTRL #OFF,DLY 0,DST 1}
DECL GRP_TYP GGDAT14={G_APO #NO,TIME 0.200000003,CTRL #OFF,DLY 0,DST 1}
DECL GRP_TYP GGDAT15={G_APO #NO,TIME 0.200000003,CTRL #OFF,DLY 0,DST 1}
DECL GRP_TYP GGDAT16={G_APO #NO,TIME 0.200000003,CTRL #OFF,DLY 0,DST 1}
DECL E6POS XP2004={x -1057.00403,y 600.57782,z 2451.78394,a 175.840302,b -72.5612793,c 179.208603,s 2,t 3,e1 0.0,e2 0.0,e3 0.0,e4 0.0,e5 0.0,e6 0.0}
DECL FDAT Fp2004={TOOL_NO 3,BASE_NO 0,IPO_FRAME #BASE}
DECL PDAT PPDAT53={VEL 100.0,ACC 100.0,APO_DIST 10.0}
DECL E6POS XP2005={x -1056.98401,y 600.554688,z 2451.80591,a 175.844696,b -72.5621872,c 179.204498,s 2,t 3,e1 0.0,e2 0.0,e3 0.0,e4 0.0,e5 0.0,e6 0.0}
DECL FDAT Fp2005={TOOL_NO 3,BASE_NO 0,IPO_FRAME #BASE}
DECL PDAT PPDAT54={VEL 100.0,ACC 100.0,APO_DIST 10.0}
ENDDAT
